VAR_GLOBAL
	xSystemOverrideMode : BOOL; (* Global system override for the prototype section*)
END_VAR

(* stored: Version 1.1.0.1, ProductVersion 3.1.4022.12
   GVL GVL_VARIABLES: Id {f5eb425e-877f-4a98-b4fc-8b7970a753e9} *)
